FUNCTION_BLOCK Wrapper_produce (* Basic Function Block Type *)
  (* Standard: 61499-2 *)
  (* Version 0.0, 5/13/2019, erik, nxtControl GmbH, Template *)
  PACKAGE Main;
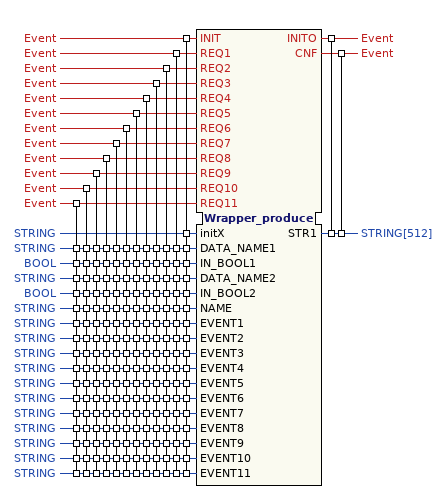
  EVENT_INPUT
    INIT WITH initX, DATA_NAME1, IN_BOOL1, DATA_NAME2, IN_BOOL2, NAME, EVENT1, EVENT2, EVENT3, EVENT4, EVENT5, EVENT6, EVENT7, EVENT8, EVENT9, EVENT10, EVENT11; (* Initialization Request *)
    REQ1 WITH DATA_NAME1, IN_BOOL1, DATA_NAME2, IN_BOOL2, NAME, EVENT1, EVENT2, EVENT3, EVENT4, EVENT5, EVENT6, EVENT7, EVENT8, EVENT9, EVENT10, EVENT11; (* Normal Execution Request *)
    REQ2 WITH DATA_NAME1, IN_BOOL1, DATA_NAME2, IN_BOOL2, NAME, EVENT1, EVENT2, EVENT3, EVENT4, EVENT5, EVENT6, EVENT7, EVENT8, EVENT9, EVENT10, EVENT11;
    REQ3 WITH DATA_NAME1, IN_BOOL1, DATA_NAME2, IN_BOOL2, NAME, EVENT1, EVENT2, EVENT3, EVENT4, EVENT5, EVENT6, EVENT7, EVENT8, EVENT9, EVENT10, EVENT11;
    REQ4 WITH DATA_NAME1, IN_BOOL1, DATA_NAME2, IN_BOOL2, NAME, EVENT1, EVENT2, EVENT3, EVENT4, EVENT5, EVENT6, EVENT7, EVENT8, EVENT9, EVENT10, EVENT11;
    REQ5 WITH DATA_NAME1, IN_BOOL1, DATA_NAME2, IN_BOOL2, NAME, EVENT1, EVENT2, EVENT3, EVENT4, EVENT5, EVENT6, EVENT7, EVENT8, EVENT9, EVENT10, EVENT11;
    REQ6 WITH DATA_NAME1, IN_BOOL1, DATA_NAME2, IN_BOOL2, NAME, EVENT1, EVENT2, EVENT3, EVENT4, EVENT5, EVENT6, EVENT7, EVENT8, EVENT9, EVENT10, EVENT11;
    REQ7 WITH DATA_NAME1, IN_BOOL1, DATA_NAME2, IN_BOOL2, NAME, EVENT1, EVENT2, EVENT3, EVENT4, EVENT5, EVENT6, EVENT7, EVENT8, EVENT9, EVENT10, EVENT11;
    REQ8 WITH DATA_NAME1, IN_BOOL1, DATA_NAME2, IN_BOOL2, NAME, EVENT1, EVENT2, EVENT3, EVENT4, EVENT5, EVENT6, EVENT7, EVENT8, EVENT9, EVENT10, EVENT11;
    REQ9 WITH DATA_NAME1, IN_BOOL1, DATA_NAME2, IN_BOOL2, NAME, EVENT1, EVENT2, EVENT3, EVENT4, EVENT5, EVENT6, EVENT7, EVENT8, EVENT9, EVENT10, EVENT11;
    REQ10 WITH DATA_NAME1, IN_BOOL1, DATA_NAME2, IN_BOOL2, NAME, EVENT1, EVENT2, EVENT3, EVENT4, EVENT5, EVENT6, EVENT7, EVENT8, EVENT9, EVENT10, EVENT11;
    REQ11 WITH DATA_NAME1, IN_BOOL1, DATA_NAME2, IN_BOOL2, NAME, EVENT1, EVENT2, EVENT3, EVENT4, EVENT5, EVENT6, EVENT7, EVENT8, EVENT9, EVENT10, EVENT11;
  END_EVENT
  EVENT_OUTPUT
    INITO WITH STR1; (* Initialization Confirm *)
    CNF WITH STR1; (* Execution Confirmation *)
  END_EVENT
  VAR_INPUT
    initX : STRING;
    DATA_NAME1 : STRING;
    IN_BOOL1 : BOOL; (* Input event qualifier *)
    DATA_NAME2 : STRING;
    IN_BOOL2 : BOOL;
    NAME : STRING;
    EVENT1 : STRING;
    EVENT2 : STRING;
    EVENT3 : STRING;
    EVENT4 : STRING;
    EVENT5 : STRING;
    EVENT6 : STRING;
    EVENT7 : STRING;
    EVENT8 : STRING;
    EVENT9 : STRING;
    EVENT10 : STRING;
    EVENT11 : STRING;
  END_VAR
  VAR_OUTPUT
    STR1 : STRING[512]; (* Output event qualifier *)
  END_VAR
  VAR
    text1 : STRING[255];
  END_VAR
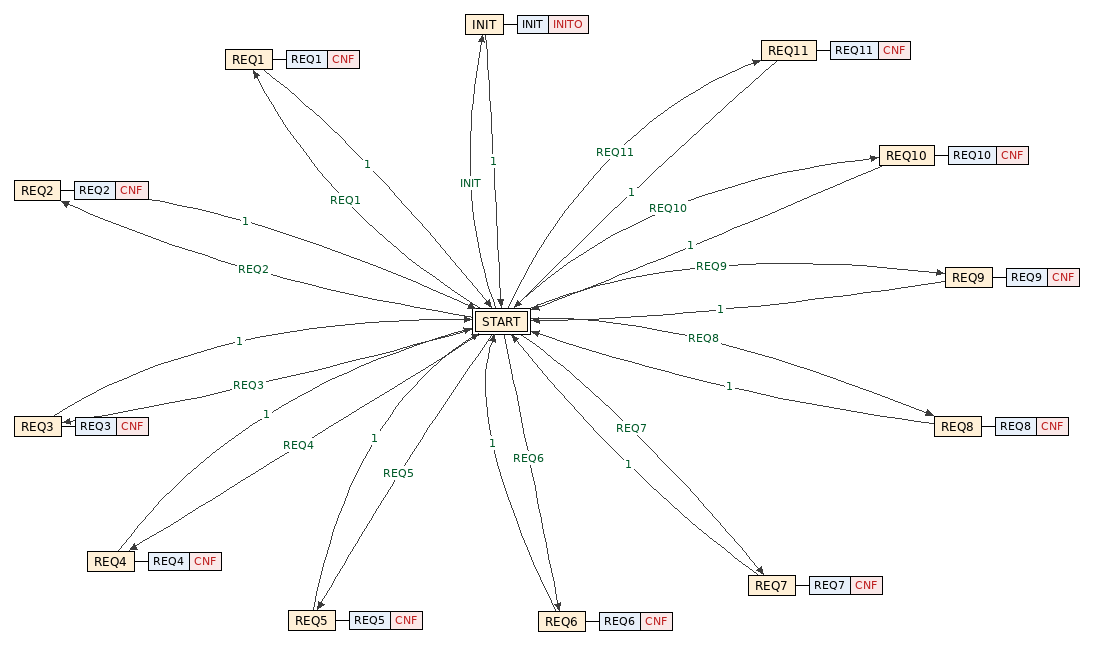
  EC_STATES
    START; (* Initial State *)
    INIT : INIT -> INITO; (* Initialization *)
    REQ1 : REQ1 -> CNF; (* Normal execution *)
    REQ2 : REQ2 -> CNF;
    REQ3 : REQ3 -> CNF;
    REQ4 : REQ4 -> CNF;
    REQ5 : REQ5 -> CNF;
    REQ6 : REQ6 -> CNF;
    REQ7 : REQ7 -> CNF;
    REQ8 : REQ8 -> CNF;
    REQ9 : REQ9 -> CNF;
    REQ10 : REQ10 -> CNF;
    REQ11 : REQ11 -> CNF;
  END_STATES
  EC_TRANSITIONS
    START TO INIT := INIT;
    INIT TO START := 1;
    START TO REQ1 := REQ1;
    REQ1 TO START := 1;
    REQ2 TO START := 1;
    START TO REQ2 := REQ2;
    REQ3 TO START := 1;
    START TO REQ3 := REQ3;
    REQ4 TO START := 1;
    START TO REQ4 := REQ4;
    REQ5 TO START := 1;
    START TO REQ5 := REQ5;
    REQ6 TO START := 1;
    START TO REQ6 := REQ6;
    REQ7 TO START := 1;
    START TO REQ7 := REQ7;
    REQ8 TO START := 1;
    START TO REQ8 := REQ8;
    REQ9 TO START := 1;
    START TO REQ9 := REQ9;
    REQ10 TO START := 1;
    START TO REQ10 := REQ10;
    REQ11 TO START := 1;
    START TO REQ11 := REQ11;
  END_TRANSITIONS
  ALGORITHM INIT IN ST: (* Initialization algorithm *)
VAR
  events : STRING[255];
  data : STRING[255];
  len1 : DINT;
END_VAR


events := '';
data := '';



(*initX is the type of init and IN_STR1 is the name*)
STR1 := initX;
STR1 := CONCAT(STR1,';');
STR1 := CONCAT(STR1,NAME);
STR1 := CONCAT(STR1,';');


IF EVENT1 <> '' THEN
	events := CONCAT(events,EVENT1);
	events := CONCAT(events,':');
END_IF;
IF EVENT2 <> '' THEN
	events := CONCAT(events,EVENT2);
	events := CONCAT(events,':');
END_IF;
IF EVENT3 <> '' THEN
	events := CONCAT(events,EVENT3);
	events := CONCAT(events,':');
END_IF;
IF EVENT4 <> '' THEN
	events := CONCAT(events,EVENT4);
	events := CONCAT(events,':');
END_IF;
IF EVENT5 <> '' THEN
	events := CONCAT(events,EVENT5);
	events := CONCAT(events,':');
END_IF;
IF EVENT6 <> '' THEN
  events := CONCAT(events,EVENT6);
  events := CONCAT(events,':');
END_IF;
IF EVENT7 <> '' THEN
  events := CONCAT(events,EVENT7);
  events := CONCAT(events,':');
END_IF;
IF EVENT8 <> '' THEN
  events := CONCAT(events,EVENT8);
  events := CONCAT(events,':');
END_IF;
IF EVENT9 <> '' THEN
  events := CONCAT(events,EVENT9);
  events := CONCAT(events,':');
END_IF;
IF EVENT10 <> '' THEN
  events := CONCAT(events,EVENT10);
  events := CONCAT(events,':');
END_IF;
IF EVENT11 <> '' THEN
  events := CONCAT(events,EVENT11);
  events := CONCAT(events,':');
END_IF;
IF events <> '' THEN
	len1 := LEN(events);
	events := LEFT(events, len1 -1);
END_IF;
events := CONCAT(events, ';');

(*joining the events to the STR1*)
STR1 := CONCAT(STR1, events);



(*data*)
data := '';
IF DATA_NAME1 <> '' THEN
	data := CONCAT(data,DATA_NAME1);
	data := CONCAT(data,':');
END_IF;
IF DATA_NAME2 <> '' THEN
  data := CONCAT(data,DATA_NAME2);
  data := CONCAT(data,':');
END_IF;
IF data <> '' THEN
	len1 := LEN(data);
	data := LEFT(data, len1 -1);
END_IF;

data := CONCAT(data, ';');


(*joining data to STR1*)
STR1 := CONCAT(STR1,data);
  END_ALGORITHM
  ALGORITHM REQ1 IN ST: (* Normally executed algorithm *)
;


STR1 := CONCAT('update;',NAME);
STR1 := CONCAT(STR1,';');

STR1 := CONCAT(STR1,EVENT1);
STR1 := CONCAT(STR1,';');

STR1 := CONCAT(STR1,'None');

STR1 := CONCAT(STR1,';');
  END_ALGORITHM
  ALGORITHM REQ2 IN ST:
;
STR1 := CONCAT('update;',NAME);
STR1 := CONCAT(STR1,';');

STR1 := CONCAT(STR1,EVENT2);
STR1 := CONCAT(STR1,';');

STR1 := CONCAT(STR1,'None');

STR1 := CONCAT(STR1,';');
  END_ALGORITHM
  ALGORITHM REQ3 IN ST:
;
STR1 := CONCAT('update;',NAME);
STR1 := CONCAT(STR1,';');

STR1 := CONCAT(STR1,EVENT3);
STR1 := CONCAT(STR1,';');

STR1 := CONCAT(STR1,'None');

STR1 := CONCAT(STR1,';');
  END_ALGORITHM
  ALGORITHM REQ4 IN ST:
;
STR1 := CONCAT('update;',NAME);
STR1 := CONCAT(STR1,';');

STR1 := CONCAT(STR1,EVENT4);
STR1 := CONCAT(STR1,';');

STR1 := CONCAT(STR1,'None');

STR1 := CONCAT(STR1,';');
  END_ALGORITHM
  ALGORITHM REQ5 IN ST:
;
STR1 := CONCAT('update;',NAME);
STR1 := CONCAT(STR1,';');

STR1 := CONCAT(STR1,EVENT5);
STR1 := CONCAT(STR1,';');

STR1 := CONCAT(STR1,'None');

STR1 := CONCAT(STR1,';');
  END_ALGORITHM
  ALGORITHM REQ6 IN ST:
;
STR1 := CONCAT('update;',NAME);
STR1 := CONCAT(STR1,';');

STR1 := CONCAT(STR1,EVENT6);
STR1 := CONCAT(STR1,';');

STR1 := CONCAT(STR1,'None');

STR1 := CONCAT(STR1,';');
  END_ALGORITHM
  ALGORITHM REQ7 IN ST:
;
STR1 := CONCAT('update;',NAME);
STR1 := CONCAT(STR1,';');

STR1 := CONCAT(STR1,EVENT7);
STR1 := CONCAT(STR1,';');

STR1 := CONCAT(STR1,'None');

STR1 := CONCAT(STR1,';');
  END_ALGORITHM
  ALGORITHM REQ8 IN ST:
;
STR1 := CONCAT('update;',NAME);
STR1 := CONCAT(STR1,';');

STR1 := CONCAT(STR1,EVENT8);
STR1 := CONCAT(STR1,';');

STR1 := CONCAT(STR1,'None');

STR1 := CONCAT(STR1,';');
  END_ALGORITHM
  ALGORITHM REQ9 IN ST:
;
STR1 := CONCAT('update;',NAME);
STR1 := CONCAT(STR1,';');

STR1 := CONCAT(STR1,EVENT9);
STR1 := CONCAT(STR1,';');

STR1 := CONCAT(STR1,'None');

STR1 := CONCAT(STR1,';');
  END_ALGORITHM
  ALGORITHM REQ10 IN ST:
;
STR1 := CONCAT('update;',NAME);
STR1 := CONCAT(STR1,';');

STR1 := CONCAT(STR1,EVENT10);
STR1 := CONCAT(STR1,';');

STR1 := CONCAT(STR1,'None');

STR1 := CONCAT(STR1,';');
  END_ALGORITHM
  ALGORITHM REQ11 IN ST:
;
STR1 := CONCAT('update;',NAME);
STR1 := CONCAT(STR1,';');

STR1 := CONCAT(STR1,EVENT11);
STR1 := CONCAT(STR1,';');

STR1 := CONCAT(STR1,'None');

STR1 := CONCAT(STR1,';');
  END_ALGORITHM
END_FUNCTION_BLOCK
